(* IEC 61131-3 sources: RL_MAR/experiments/comparison/llm4plc/results/gpt-4o-mini_20260506_100619/20260506_104015, 1 file *)

(* ---- generated_code_iteration_0.st ---- *)
ructured-text
FUNCTION_BLOCK SoilTestingDeviceControl
VAR_INPUT
    StartButton : BOOL; (* Input for starting the testing process *)
    SoilSampleDetected : BOOL; (* Input for detecting soil sample *)
END_VAR
VAR_OUTPUT
    NutrientPump : BOOL; (* Output to control nutrient pump *)
    pHAdjustmentPump : BOOL; (* Output to control pH adjustment pump *)
END_VAR
VAR
    pHSensorValue : REAL; (* Simulated pH sensor value *)
    NutrientSensorValue : REAL; (* Simulated nutrient sensor value *)
    TestingStatus : INT; (* Status: 0=Idle, 1=Testing, 2=Completed *)
    NutrientThreshold : REAL := 0.7; (* Nutrient level threshold for analysis *)
    pHThreshold : REAL := 6.5; (* pH level threshold for analysis *)
END_VAR

(* Initialization Logic *)
IF TestingStatus = 0 THEN
    pHSensorValue := 7.0;
    NutrientSensorValue := 0.5;
END_IF

(* Start/Testing Logic *)
IF TestingStatus = 0 AND StartButton = TRUE THEN
    TestingStatus := 1; (* Transition to Testing *)
    NutrientPump := TRUE; (* Activate Nutrient Pump *)
    pHAdjustmentPump := TRUE; (* Activate pH Adjustment Pump *)
END_IF

(* Simulated Sensor Value Updates (During Testing) *)
IF TestingStatus = 1 THEN
    IF NutrientSensorValue < 0.9 THEN
        NutrientSensorValue := NutrientSensorValue + 0.1; (* Increment Nutrient Sensor Value *)
    END_IF
    IF pHSensorValue > 4.0 THEN
        pHSensorValue := pHSensorValue - 0.5; (* Decrement pH Sensor Value *)
    END_IF

    (* Completion Logic *)
    IF SoilSampleDetected = TRUE THEN
        IF NutrientSensorValue >= NutrientThreshold AND pHSensorValue <= pHThreshold THEN
            TestingStatus := 2; (* Transition to Completed *)
            NutrientPump := FALSE; (* Deactivate Nutrient Pump *)
            pHAdjustmentPump := FALSE; (* Deactivate pH Adjustment Pump *)
        END_IF
    END_IF
END_IF

(* Optional: Reset or wait for next test logic can be added here if needed *)

END_FUNCTION_BLOCK
